DATA_BLOCK "CalcVolume_Tank14_DB"
{ S7_Optimized_Access := 'FALSE' }
VERSION : 0.1
"CalculationVolume"

BEGIN
   IW_Radius := 3.102;
   IW_ValueFromSensor := 17.18027;
   IW_K_for_Tonnag := 1.35;
   IW_K_for_Level := 1.35;
   QW_Volume := 384.5115;
   QW_Tonnag := 519.0905;
   QW_RealLevel := 12.72612;
   sW_S := 30.21435;
   sW_Volume := 384.5115;
   sW_RealLevel := 12.72612;

END_DATA_BLOCK

